TYPE TAxisHomingType :
	(	AHT_NoHoming,
		AHT_OnSensor,
		AHT_OnZeroEncoder
	);
END_TYPE

(* stored: Version 1.1.0.1, ProductVersion 3.1.4022.12
   DUT TAxisHomingType: Id {3939d4ae-6ded-44f9-870e-e2e5d55ac766} *)
